// Mitsubishi GX Works2 project: Project_3.1   PLC: Q03UDV

PROGRAM MAIN
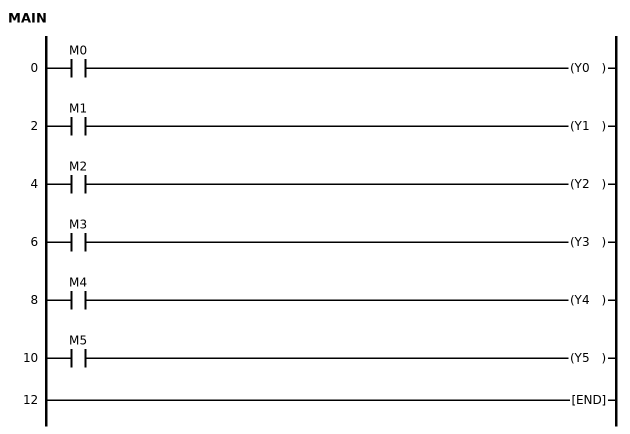
0     LD      M0
      OUT     Y0
2     LD      M1
      OUT     Y1
4     LD      M2
      OUT     Y2
6     LD      M3
      OUT     Y3
8     LD      M4
      OUT     Y4
10    LD      M5
      OUT     Y5
12    END
END_PROGRAM
